FUNCTION_BLOCK ValveMonitor
VAR_INPUT
	Valve: BOOL;	// Valve DO
	FB1: BOOL;		// Open DI
	FB2: BOOL;		// Closed DI
	Timeout: TIME;
END_VAR
VAR_OUTPUT
	Error: BOOL;
END_VAR
VAR
	ValveSignal: DigitalSignal;
	ValveOpenTimer: Timer;
	ValveClosedTimer: Timer;
END_VAR

ValveSignal(Signal := Valve);
Error := ((ValveSignal.OnTime() > TO_LINT(Timeout)) AND (NOT FB1)) OR
		((ValveSignal.OffTime() > TO_LINT(Timeout)) AND (NOT FB2));

END_FUNCTION_BLOCK

(* stored: Version 1.1.0.1, ProductVersion 3.1.4024.6
   POU ValveMonitor: Id {5e5c3826-97f3-4bfe-aef7-529bb9c4edeb}, SpecialFunc None *)
